// TIA Portal V20 export
TYPE "type_emRelations_em1_cmStatus"
// stored: Access Published, Namespace Unit1
   STRUCT
      Stacker2NgBoxDetect { S7_SetPoint := 'True'} : "LBC_typeDigitalSignalControlNode";
      Stacker2NgBoxFullDetect { S7_SetPoint := 'True'} : "LBC_typeDigitalSignalControlNode";
      Stacker2NgBoxLoadingUpDown { S7_SetPoint := 'True'} : "LBC_typeTwoWayActuatorControlNode";
      Stacker2NgBoxUnitMoverBwdFwd { S7_SetPoint := 'True'} : "LBC_typeTwoWayActuatorControlNode";
      Stacker2NgBoxClampLeftOpenClose { S7_SetPoint := 'True'} : "LBC_typeTwoWayActuatorControlNode";
      Stacker2NgBoxClampRightOpenClose { S7_SetPoint := 'True'} : "LBC_typeTwoWayActuatorControlNode";
      Stacker2NgBoxClampMoverOpenClose { S7_SetPoint := 'True'} : "LBC_typeTwoWayActuatorControlNode";
      Stacker2NgBoxLiftDownUp { S7_SetPoint := 'True'} : "LBC_typeTwoWayActuatorControlNode";
      Stacker2NgBoxLockDownUp { S7_SetPoint := 'True'} : "LBC_typeTwoWayActuatorControlNode";
   END_STRUCT;
END_TYPE
